(* Logix 5000 project; controller Almacen_2 vendor 1 type 14 code 235 rev 36.11; software revision 36.00; part 2 of 2 *)
(* tags used below, declared in another part *)
   Contador_Salida_Conveyor : COUNTER;
   End_Conveyor_Rutine : BOOL;
   Start_Conveyor_2 : BOOL;
   Start_Rutine : BOOL;
   Stop_Conveyor_2 : BOOL;
   tag_switch : BOOL;
   tag_switch2 : BOOL;
   tag_switch3 : BOOL;
   Tag_switch4 : BOOL;
   tag_switch5 : BOOL;
   tag_switch6 : BOOL;
   tag_timer_piston : BOOL;
   tag_timer_piston2 : BOOL;
   Timer1_Cambio_Direccion_CNC : TIMER;
   Timer2 : TIMER;
   Timer3_Piston_Marcadora_OFF : TIMER;
   Timer4_Piston_Camara_ON : TIMER;
   Timer5_Piston_Camara_OFF : TIMER;
   Timer6_Cambio_Direccion_Almacen : TIMER;
   Timer7_Sensor_Entrada_Salida : TIMER;
   Timer8_Stop_Conveyor : TIMER;
   Timer9_Piston_Salida : TIMER;
   At_Pos_Alm_2 : DINT;
   Estops_Ok : BOOL;
   In_Pos_Alm_2 : DINT;
   Interlocks_Ok : BOOL;
   LigthCurtain2_Ok : BOOL;
   PosicionAlmacen : DINT;
   Safety_FromTEC81 : Safety;
   Sfty_OK : BOOL;
   Start_Kinetix_Alm_2 : DINT;
   Start_Motor_Alm_2 : BOOL;
   To_Pos_Alm_2 : DINT;
(* MainProgram, continued *)

ROUTINE Movimiento_elevador_Alm_2   (* ladder *)
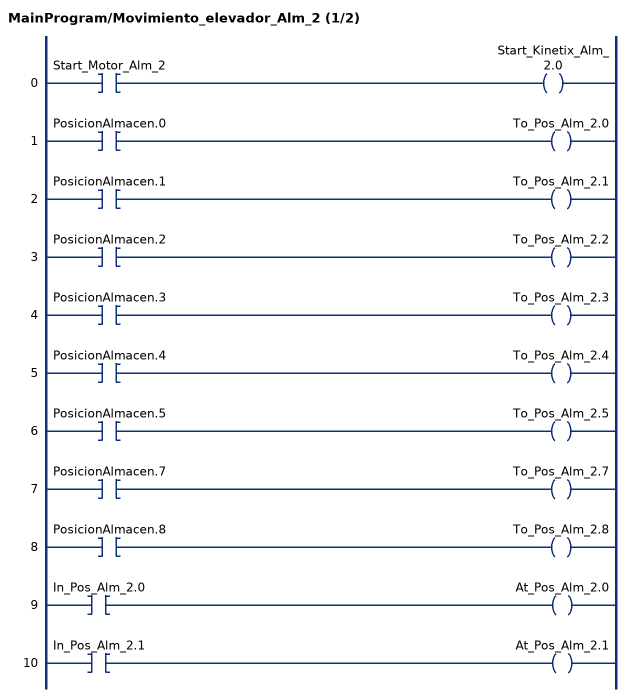
   0: XIC(Start_Motor_Alm_2)OTE(Start_Kinetix_Alm_2.0);
   1: XIC(PosicionAlmacen.0)OTE(To_Pos_Alm_2.0);
   2: XIC(PosicionAlmacen.1)OTE(To_Pos_Alm_2.1);
   3: XIC(PosicionAlmacen.2)OTE(To_Pos_Alm_2.2);
   4: XIC(PosicionAlmacen.3)OTE(To_Pos_Alm_2.3);
   5: XIC(PosicionAlmacen.4)OTE(To_Pos_Alm_2.4);
   6: XIC(PosicionAlmacen.5)OTE(To_Pos_Alm_2.5);
   7: XIC(PosicionAlmacen.7)OTE(To_Pos_Alm_2.7);
   8: XIC(PosicionAlmacen.8)OTE(To_Pos_Alm_2.8);
   9: XIC(In_Pos_Alm_2.0)OTE(At_Pos_Alm_2.0);
   10: XIC(In_Pos_Alm_2.1)OTE(At_Pos_Alm_2.1);
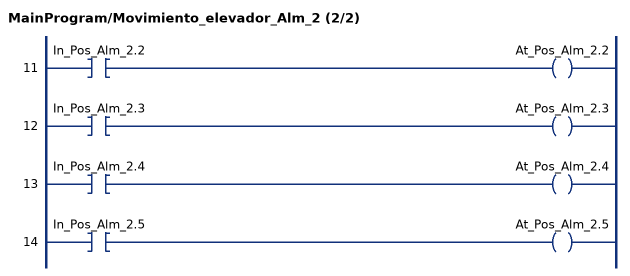
   11: XIC(In_Pos_Alm_2.2)OTE(At_Pos_Alm_2.2);
   12: XIC(In_Pos_Alm_2.3)OTE(At_Pos_Alm_2.3);
   13: XIC(In_Pos_Alm_2.4)OTE(At_Pos_Alm_2.4);
   14: XIC(In_Pos_Alm_2.5)OTE(At_Pos_Alm_2.5);
END_ROUTINE

ROUTINE Prueba   (* ladder *)
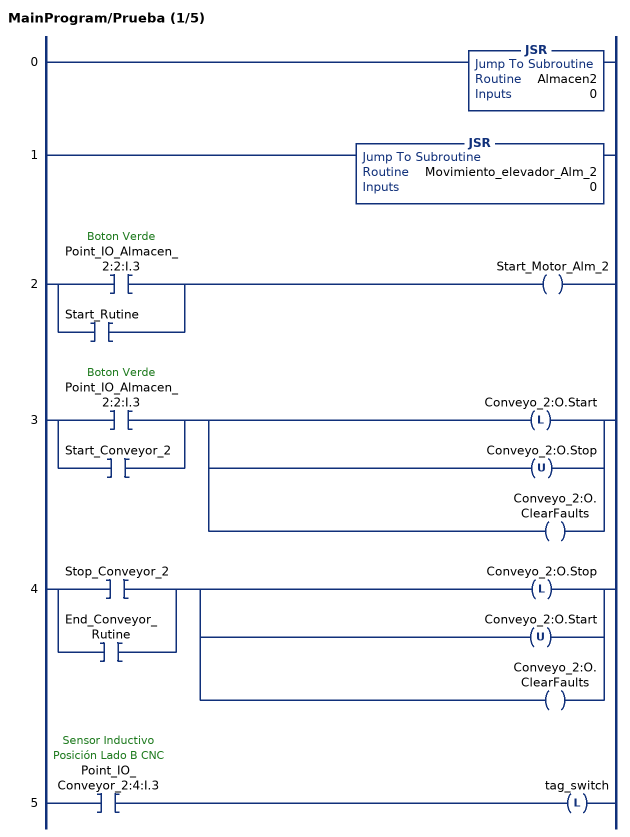
   0: JSR(Almacen2,0);
   1: JSR(Movimiento_elevador_Alm_2,0);
   2: [XIC(Point_IO_Almacen_2:2:I.3) ,XIC(Start_Rutine) ]OTE(Start_Motor_Alm_2);
   3: [XIC(Point_IO_Almacen_2:2:I.3) ,XIC(Start_Conveyor_2) ][OTL(Conveyo_2:O.Start) ,OTU(Conveyo_2:O.Stop) ,OTE(Conveyo_2:O.ClearFaults) ];
   4: [XIC(Stop_Conveyor_2) ,XIC(End_Conveyor_Rutine) ][OTL(Conveyo_2:O.Stop) ,OTU(Conveyo_2:O.Start) ,OTE(Conveyo_2:O.ClearFaults) ];
   5: XIC(Point_IO_Conveyor_2:4:I.3)OTL(tag_switch);
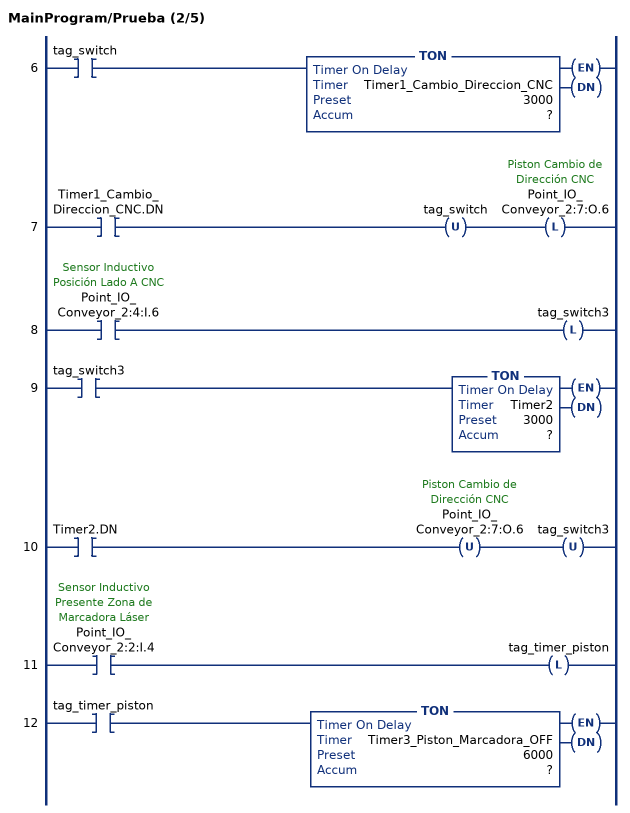
   6: XIC(tag_switch)TON(Timer1_Cambio_Direccion_CNC,?,?);
   7: XIC(Timer1_Cambio_Direccion_CNC.DN)OTU(tag_switch)OTL(Point_IO_Conveyor_2:7:O.6);
   8: XIC(Point_IO_Conveyor_2:4:I.6)OTL(tag_switch3);
   9: XIC(tag_switch3)TON(Timer2,?,?);
   10: XIC(Timer2.DN)OTU(Point_IO_Conveyor_2:7:O.6)OTU(tag_switch3);
   11: XIC(Point_IO_Conveyor_2:2:I.4)OTL(tag_timer_piston);
   12: XIC(tag_timer_piston)TON(Timer3_Piston_Marcadora_OFF,?,?);
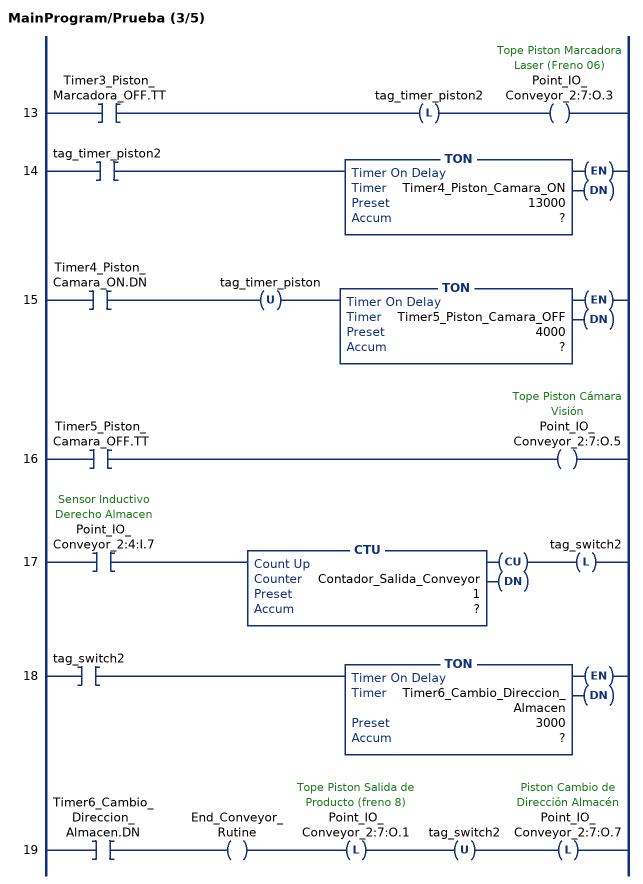
   13: XIC(Timer3_Piston_Marcadora_OFF.TT)OTL(tag_timer_piston2)OTE(Point_IO_Conveyor_2:7:O.3);
   14: XIC(tag_timer_piston2)TON(Timer4_Piston_Camara_ON,?,?);
   15: XIC(Timer4_Piston_Camara_ON.DN)OTU(tag_timer_piston)TON(Timer5_Piston_Camara_OFF,?,?);
   16: XIC(Timer5_Piston_Camara_OFF.TT)OTE(Point_IO_Conveyor_2:7:O.5);
   17: XIC(Point_IO_Conveyor_2:4:I.7)CTU(Contador_Salida_Conveyor,?,?)OTL(tag_switch2);
   18: XIC(tag_switch2)TON(Timer6_Cambio_Direccion_Almacen,?,?);
   19: XIC(Timer6_Cambio_Direccion_Almacen.DN)OTE(End_Conveyor_Rutine)OTL(Point_IO_Conveyor_2:7:O.1)OTU(tag_switch2)OTL(Point_IO_Conveyor_2:7:O.7);
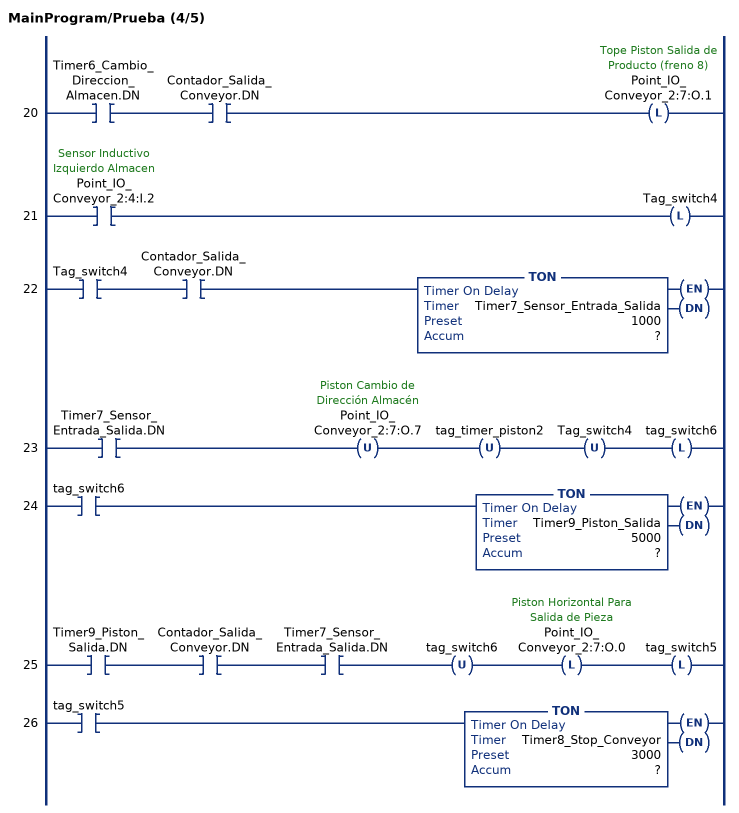
   20: XIC(Timer6_Cambio_Direccion_Almacen.DN)XIC(Contador_Salida_Conveyor.DN)OTL(Point_IO_Conveyor_2:7:O.1);
   21: XIC(Point_IO_Conveyor_2:4:I.2)OTL(Tag_switch4);
   22: XIC(Tag_switch4)XIC(Contador_Salida_Conveyor.DN)TON(Timer7_Sensor_Entrada_Salida,?,?);
   23: XIC(Timer7_Sensor_Entrada_Salida.DN)OTU(Point_IO_Conveyor_2:7:O.7)OTU(tag_timer_piston2)OTU(Tag_switch4)OTL(tag_switch6);
   24: XIC(tag_switch6)TON(Timer9_Piston_Salida,?,?);
   25: XIC(Timer9_Piston_Salida.DN)XIC(Contador_Salida_Conveyor.DN)XIC(Timer7_Sensor_Entrada_Salida.DN)OTU(tag_switch6)OTL(Point_IO_Conveyor_2:7:O.0)OTL(tag_switch5);
   26: XIC(tag_switch5)TON(Timer8_Stop_Conveyor,?,?);
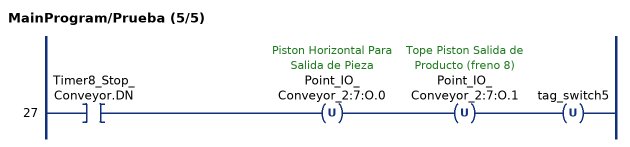
   27: XIC(Timer8_Stop_Conveyor.DN)OTU(Point_IO_Conveyor_2:7:O.0)OTU(Point_IO_Conveyor_2:7:O.1)OTU(tag_switch5);
END_ROUTINE
END_PROGRAM

PROGRAM SafetyProgram   (* main routine MainRoutine, safety *)

ROUTINE External_COMM   (* ladder *)
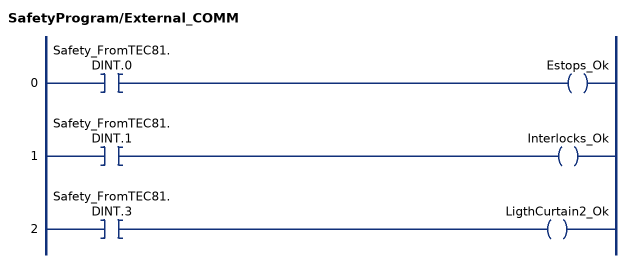
   0: XIC(Safety_FromTEC81.DINT.0)OTE(Estops_Ok);
   1: XIC(Safety_FromTEC81.DINT.1)OTE(Interlocks_Ok);
   2: XIC(Safety_FromTEC81.DINT.3)OTE(LigthCurtain2_Ok);
END_ROUTINE

ROUTINE MainRoutine   (* ladder *)
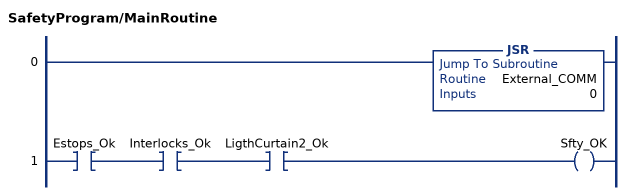
   0: JSR(External_COMM,0);
   1: XIC(Estops_Ok)XIC(Interlocks_Ok)XIC(LigthCurtain2_Ok)OTE(Sfty_OK);
END_ROUTINE
END_PROGRAM
